FUNCTION_BLOCK Test
VAR_INPUT
END_VAR
VAR_OUTPUT
END_VAR
VAR
END_VAR

METHOD Wait1S : BOOL
VAR_INPUT
END_VAR
END_METHOD

END_FUNCTION_BLOCK

(* stored: Version 1.1.0.1, ProductVersion 3.1.4026.18
   POU Test: Id {afa0652a-0b0e-439a-895a-1524d428d0d9}, SpecialFunc None
   Method Wait1S: Id {e566fc96-555b-4d49-9612-f8e0c62b01f1} *)
